PROGRAM MAIN
VAR
	HS AT %I*:BOOL;
	DataHoraIHM:DATE_AND_TIME;
	testeString:STRING;
	NomeUsuario:STRING;		//Nome do usuário vindo da IHM
	SerialDaMaquina:STRING;		//Serial da máquina com 16 digitos
	
	//Reloj
	fbTime: FB_LocalSystemTime;
	DataHora	:STRING;
	wHora		:INT;
	wMin		: INT;
	wSec		: INT;


	indice: INT;
	SetLocalTime: NT_SetLocalTime;	//Instância para ajustar a hora
	
	Teste:UDINT;
	Teste2:time;
	Teste3:DT;
	fbSystemTime : GETSYSTEMTIME;
    timeAsFileTime : T_FILETIME;
	
	
	HoraAtual	:DT;	//Hora atual
	udHoraAtual	:UDINT;	//Hora atual em UDINT
	// variavel para testes
	i: INT;
END_VAR

//Serial da máquina
SerialDaMaquina := 'LS-B300S-001';



//Ajusta a data e hora do CLP pela IHM
SetLocalTime(
	NETID:= '127.0.0.1.1.1', 
	TIMESTR:= , 
	START:= , 
	TMOUT:= , 
	BUSY=> , 
	ERR=> , 
	ERRID=> );
IF SetLocalTime.START THEN
	SetLocalTime.START := FALSE;
END_IF

//Essa parte do código é utilizada para auxiliar na verificação da útima vez da calibração/lavagem 
fbSystemTime(
    timeLoDW=>timeAsFileTime.dwLowDateTime,
    timeHiDW=>timeAsFileTime.dwHighDateTime 
);

HoraAtual 	:= FILETIME_TO_DT(timeAsFileTime); 
udHoraAtual	:= DT_TO_UDINT(HoraAtual);

Teste := TIME_TO_UDINT(t#1D);



//'DT#1970-01-01-00:00:00'
SetLocalTime.TIMESTR.wDay		:= STRING_TO_WORD(MID(DT_TO_STRING(DataHoraIHM), 2, 12));
SetLocalTime.TIMESTR.wMonth		:= STRING_TO_WORD(MID(DT_TO_STRING(DataHoraIHM), 2, 9));
SetLocalTime.TIMESTR.wYear		:= STRING_TO_WORD(MID(DT_TO_STRING(DataHoraIHM), 4, 4));
SetLocalTime.TIMESTR.wHour		:= STRING_TO_WORD(MID(DT_TO_STRING(DataHoraIHM - T#3H), 2, 15));
SetLocalTime.TIMESTR.wMinute	:= STRING_TO_WORD(MID(DT_TO_STRING(DataHoraIHM), 2, 18));
SetLocalTime.TIMESTR.wSecond	:= STRING_TO_WORD(MID(DT_TO_STRING(DataHoraIHM), 2, 21));

//Faz a leitura da data e hora
fbTime(
	sNetID:= '' , 
	bEnable:= TRUE, 
	dwCycle:=1 , 
	dwOpt:= , 
	tTimeout:= , 
	bValid=> , 
	systemTime=> , 
	tzID=> );
wHora:=WORD_TO_INT(fbTime.systemTime.wHour);
wMin:=WORD_TO_INT(fbTime.systemTime.wMinute);
wSec:=WORD_TO_INT(fbTime.systemTime.wSecond);


//Data e hora formatada para a IHM
//dd/MM/AAAA, HH:mm
DataHora := CONCAT(
    CONCAT(
        CONCAT(
            CONCAT(
                CONCAT(
                    WORD_TO_STRING(fbTime.systemTime.wDay), '/'
                ),
                WORD_TO_STRING(fbTime.systemTime.wMonth)
            ),
            '/'
        ),
        WORD_TO_STRING(fbTime.systemTime.wYear)
    ),
    CONCAT(
        CONCAT(', ', INT_TO_STRING(wHora)),
        CONCAT(':', INT_TO_STRING(wMin))
    )
);

//Inicializacion de variables
IF HMI.iCircuito_a_calibrar=0 THEN
	HMI.iCircuito_a_calibrar:=1;
END_IF
FOR indice:= 1 TO 12 BY 1 DO
	IF Liquidos.Circuito_Liquido[indice]=0 THEN
		Liquidos.Circuito_Liquido[indice]:=1;
	END_IF
END_FOR

//Verifica se tem alguma linha de pó sem produto definido
FOR indice := 1 TO 4 DO
	IF Polvos.ProdutoAsociado[indice] = 0 THEN
		Polvos.ProdutoAsociado[indice] := 1;
	END_IF
END_FOR


VarPersistentes();
Datos_Variadores();
Datos_Caudalimetros();
Agitadores();
_Seguridad();
Alarmas();
Inicio();
Tratadora();
Balanza_Semilla();
Puesto_CA1();
Circuito_L1();
Circuito_L2();
Circuito_L3();
Circuito_L4();
Puesto_CA2();
Circuito_L5();
Circuito_L6();
Circuito_L7();
Circuito_L8();
Puesto_CA3();
Circuito_L9();
Circuito_L10();
Circuito_L11();
Circuito_L12();
Valvulas_Lavado();
Dosificador_Polvo_1();
Dosificador_Polvo_2();
Carga_Semilla();
Descarga_Semilla();

//Testes
Receitas();
PRG_DE_TESTES();
//BancoDeDados();
AlarmesDaMaquina();
IntervaloLavCalibr();
CalculoConsumo();
ConsumoIBCs();
AquecimentoValvulas();
ConfigBombas();
iPC_Diagnostic();

END_PROGRAM

(* stored: Version 1.1.0.1, ProductVersion 3.1.4024.14
   POU MAIN: Id {7203522a-8804-4c33-8a85-aa46ba3fd22d}, SpecialFunc None *)
